FUNCTION_BLOCK PTRC_Logic (* Basic Function Block Type *)
  (* Standard: 61499-2 *)
  (* Version 0.0, 12/10/2023, Cheyan, Schneider Electric, Template *)
  PACKAGE Main;
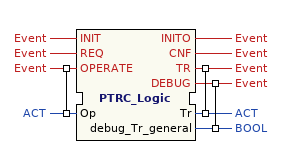
  EVENT_INPUT
    INIT; (* Initialization Request *)
    REQ; (* Normal Execution Request *)
    OPERATE WITH Op;
  END_EVENT
  EVENT_OUTPUT
    INITO; (* Initialization Confirm *)
    CNF; (* Execution Confirmation *)
    TR WITH Tr;
    DEBUG WITH debug_Tr_general;
  END_EVENT
  VAR_INPUT
    Op : ACT; (* Input event qualifier *)
  END_VAR
  VAR_OUTPUT
    Tr : ACT; (* Output event qualifier *)
    debug_Tr_general : BOOL;
  END_VAR
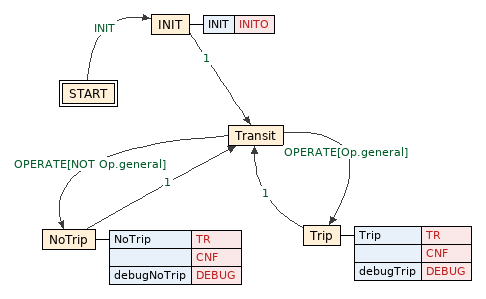
  EC_STATES
    START; (* Initial State *)
    INIT : INIT -> INITO; (* Initialization *)
    Trip : Trip -> TR, -> CNF, debugTrip -> DEBUG; (* Normal execution *)
    Transit;
    NoTrip : NoTrip -> TR, -> CNF, debugNoTrip -> DEBUG;
  END_STATES
  EC_TRANSITIONS
    START TO INIT := INIT;
    INIT TO Transit := 1;
    Transit TO Trip := OPERATE[Op.general];
    Trip TO Transit := 1;
    Transit TO NoTrip := OPERATE[NOT Op.general];
    NoTrip TO Transit := 1;
  END_TRANSITIONS
  ALGORITHM INIT IN ST: (* Initialization algorithm *)
;
  END_ALGORITHM
  ALGORITHM Trip IN ST: (* Normally executed algorithm When the trip condition is met (i.e. overcurrent fault is detected), Tr_general is set to TRUE. *)
;

Tr.general := TRUE;
  END_ALGORITHM
  ALGORITHM NoTrip IN ST:
;

Tr.general := FALSE;
  END_ALGORITHM
  ALGORITHM debugTrip IN ST:
;

debug_Tr_general := TRUE;
  END_ALGORITHM
  ALGORITHM debugNoTrip IN ST:
;

debug_Tr_general := FALSE;
  END_ALGORITHM
END_FUNCTION_BLOCK
